SUBAPPLICATION Uebung_171 (* Exercise for E_D_FF_ANY *)
  (* Standard: 61499-2; Description: Copyright (c) 2023 Meisterschulen am Ostbahnhof This program and the accompanying materials are made available under the terms of the Eclipse Public License 2.0 which is available at https://www.eclipse.org/legal/epl-2.0/ SPDX-License-Identifier: EPL-2.0 *)
  (* Version 1.0, 2025-02-01, Franz Höpfinger, Meisterschulen am Ostbahnhof, initial API and implementation and/or initial documentation *)
  PACKAGE Uebungen;
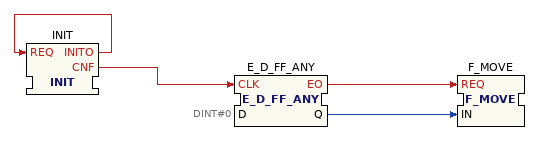
  (* E_D_FF_ANY ist eine "Event Bremse" die nur weiterleitet wenn sich D geändert hat. *)
  FBS
    E_D_FF_ANY : iec61499::events::E_D_FF_ANY(D := DINT#0);
    F_MOVE : iec61131::selection::F_MOVE; {SET_ATTRIBUTE(DataType, DINT)}
    INIT : iec61131::booleanOperators::INIT;
  END_FBS
  EVENT_CONNECTIONS
    E_D_FF_ANY.EO TO F_MOVE.REQ;
    INIT.INITO TO INIT.REQ;
    INIT.CNF TO E_D_FF_ANY.CLK;
  END_CONNECTIONS
  DATA_CONNECTIONS
    E_D_FF_ANY.Q TO F_MOVE.IN;
  END_CONNECTIONS
END_SUBAPPLICATION
